Yaskawa INFORM job: OK_R2_O55B(90,0)KMOK.JBI

/JOB
//NAME OK_R2_O55B(90,0)KMOK
//POS
///NPOS 392,392,392,17,0,0
///TOOL 0
///POSTYPE PULSE
///PULSE
C00000=10240,-83405,-67778,-29541,62233,41875
C00001=74443,53482,-30,-19359,82189,66632
C00002=132592,-56559,-52251,-28632,66053,40913
C00003=129345,-24135,-32044,-25757,67809,37971
C00004=128077,-19433,-26422,-25478,66476,37777
C00005=126545,-19710,-26626,-24916,65999,37273
C00006=128077,-19433,-26422,-25478,66476,37777
C00007=128077,-19205,-24592,-25664,65564,37989
C00008=128077,-19433,-26422,-25478,66476,37777
C00009=127855,-14483,-22733,-25349,66655,37648
C00010=128077,-19433,-26422,-25478,66476,37777
C00011=128831,-22488,-30680,-25570,67657,37802
C00012=131328,-25866,-35393,-26270,69484,38362
C00013=105362,-34489,-43309,25691,63108,24690
C00014=105506,-28668,-33620,26305,60379,24076
C00015=105705,-24608,-28573,26473,59398,23909
C00016=105689,-24392,-27343,26648,58825,23753
C00017=105705,-24608,-28573,26473,59398,23909
C00018=105942,-21948,-26691,26312,59510,24040
C00019=105705,-24608,-28573,26473,59398,23909
C00020=105810,-30681,-34237,26332,59694,24030
C00021=105674,-36363,-40882,26105,60791,24250
C00022=103128,-59362,-53746,28284,58232,22422
C00023=131703,-20648,-10182,-29245,58174,41475
C00024=129196,-16533,-4757,-28754,56230,40918
C00025=126149,-3315,1827,-22038,65549,35319
C00026=126149,-2778,3575,-22172,64804,35468
C00027=126149,-3315,1827,-22038,65549,35319
C00028=124687,-3514,1666,-21646,65158,34817
C00029=126149,-3315,1827,-22038,65549,35319
C00030=126037,287,4808,-22006,65537,35277
C00031=127852,-16066,-3331,-28477,55208,40605
C00032=128831,-17793,-5581,-28669,55981,40825
C00033=131353,-23689,-16621,-28452,60169,40750
C00034=105306,-30907,-23656,28514,53942,22215
C00035=105451,-24787,-16501,28889,52781,21931
C00036=105748,-19475,-10296,29156,51720,21741
C00037=105748,-19067,-9029,29374,51220,21580
C00038=105748,-19475,-10296,29156,51720,21741
C00039=105922,-17726,-9011,29036,51756,21835
C00040=105748,-19475,-10296,29156,51720,21741
C00041=105734,-26360,-16311,29101,51869,21782
C00042=105596,-32543,-23465,28716,52996,22066
C00043=103146,-52240,-31759,31823,49615,19688
C00044=131717,-20532,-10041,-29258,58155,41487
C00045=129210,-16415,-4611,-28768,56209,40930
C00046=125726,-5717,1203,-22571,62030,35720
C00047=124600,-5859,1089,-22225,61721,35324
C00048=125726,-5717,1203,-22571,62030,35720
C00049=125726,-5303,2500,-22688,61489,35835
C00050=125726,-5717,1203,-22571,62030,35720
C00051=125653,-3254,3200,-22541,62045,35686
C00052=125726,-5717,1203,-22571,62030,35720
C00053=128784,-17293,-5015,-28681,55885,40832
C00054=131298,-23300,-16397,-28418,60205,40716
C00055=105773,-31038,-23538,28349,53659,22349
C00056=105903,-24906,-16379,28733,52505,22061
C00057=106236,-19176,-10156,28906,51612,21944
C00058=106236,-18582,-8321,29223,50886,21716
C00059=106236,-18920,-9354,29043,51293,21845
C00060=106398,-17216,-8100,28928,51328,21935
C00061=106236,-18920,-9354,29043,51293,21845
C00062=105990,-26237,-16432,28932,51901,21915
C00063=105862,-32413,-23583,28545,53028,22202
C00064=103178,-48551,-23153,33432,46714,18598
C00065=131682,-20111,-9683,-29247,58140,41477
C00066=129184,-15990,-4240,-28763,56191,40923
C00067=127040,-1088,4742,-24560,65175,37666
C00068=126467,-11690,524,-28007,54635,40139
C00069=127531,-11511,663,-28398,54998,40520
C00070=127531,-11067,1898,-28573,54527,40663
C00071=127531,-11511,663,-28398,54998,40520
C00072=127446,-9507,2221,-28343,55032,40470
C00073=127531,-11511,663,-28398,54998,40520
C00074=128904,-17444,-5156,-28721,55934,40872
C00075=131423,-23616,-17139,-28383,60508,40687
C00076=105688,-30684,-23416,28352,53783,22346
C00077=105820,-24560,-16252,28734,52622,22058
C00078=106057,-19692,-10280,29061,51509,21823
C00079=106057,-19242,-8894,29301,50963,21649
C00080=106057,-19692,-10280,29061,51509,21823
C00081=106259,-17596,-8740,28917,51554,21935
C00082=106057,-19692,-10280,29061,51509,21823
C00083=106034,-26290,-16352,28940,51819,21911
C00084=105908,-32471,-23505,28552,52945,22198
C00085=103240,-57430,-47340,29139,55590,21702
C00086=131680,-19875,-9302,-29279,58038,41504
C00087=129182,-15746,-3847,-28798,56088,40952
C00088=127763,-11793,120,-28421,55243,40554
C00089=127763,-11187,1809,-28663,54602,40747
C00090=127763,-11793,120,-28421,55243,40554
C00091=126428,-12019,-55,-27932,54786,40076
C00092=127763,-11793,120,-28421,55243,40554
C00093=127667,-9572,1845,-28358,55279,40497
C00094=127763,-11793,120,-28421,55243,40554
C00095=128878,-17535,-5369,-28685,55999,40840
C00096=131397,-24246,-19366,-28107,61425,40422
C00097=105596,-30428,-23258,28382,53845,22322
C00098=105731,-24307,-16087,28765,52679,22032
C00099=105964,-19427,-9965,29125,51490,21773
C00100=105964,-19008,-8676,29352,50979,21612
C00101=105964,-19427,-9965,29125,51490,21773
C00102=106146,-17563,-8595,28999,51530,21874
C00103=105964,-19427,-9965,29125,51490,21773
C00104=106055,-26245,-16306,28933,51808,21917
C00105=103176,-54287,-36697,30953,51210,20316
C00106=103176,-54287,-36697,30953,51210,20316
C00107=114756,-19958,-23748,4768,67559,29134
C00108=116139,-18803,-17118,-4242,63507,29437
C00109=122978,-12099,-10750,-16592,66093,31815
C00110=122978,-11495,-8359,-16737,64980,31977
C00111=122982,-12162,-10065,-16649,65658,31878
C00112=121832,-12217,-10107,-16291,65423,31469
C00113=122988,-12906,-11150,-16616,65934,31840
C00114=123134,-22680,-18382,-16732,65415,31972
C00115=117879,-24479,-16681,-8596,59721,23409
C00116=117904,-23072,-15686,-8596,59834,23409
C00117=118573,-28074,-21596,-8764,60960,23581
C00118=139843,-43230,-38559,-29857,68480,-19080
C00119=155576,-42864,-35821,-41350,65515,-28225
C00120=156680,-25452,-21834,-49402,55441,-44843
C00121=157625,-11795,-9945,-68294,73257,-47337
C00122=155300,-9623,-5312,-68606,71014,-46888
C00123=154236,-7511,-1206,-68991,69742,-46386
C00124=154236,-7054,266,-69215,69486,-46084
C00125=154236,-7511,-1206,-68991,69742,-46386
C00126=153910,-5990,11,-68964,69537,-46444
C00127=154236,-7511,-1206,-68991,69742,-46386
C00128=156732,-10707,-4701,-68974,71616,-46273
C00129=159088,-12866,-9320,-68642,73874,-46723
C00130=157785,-12020,-9831,-68356,73290,-47233
C00131=155455,-9843,-5195,-68673,71046,-46784
C00132=154312,-7370,-806,-69053,69723,-46297
C00133=154312,-6958,503,-69250,69494,-46028
C00134=154312,-7370,-806,-69053,69723,-46297
C00135=153965,-5762,476,-69025,69507,-46359
C00136=154312,-7370,-806,-69053,69723,-46297
C00137=156851,-10510,-4837,-68926,71768,-46340
C00138=159204,-12645,-9439,-68604,74024,-46790
C00139=157690,-12072,-10010,-68326,73260,-47284
C00140=155360,-9896,-5377,-68641,71015,-46835
C00141=154250,-7627,-1259,-69001,69740,-46371
C00142=154250,-7165,219,-69222,69483,-46066
C00143=154250,-7627,-1259,-69001,69740,-46371
C00144=153893,-5954,78,-68966,69513,-46438
C00145=154250,-7627,-1259,-69001,69740,-46371
C00146=156734,-10980,-5063,-68950,71650,-46310
C00147=159094,-13131,-9672,-68622,73909,-46758
C00148=157604,-12431,-10269,-68326,73193,-47285
C00149=155270,-10247,-5634,-68640,70946,-46837
C00150=154185,-8119,-1688,-68996,69699,-46385
C00151=154185,-7714,-386,-69193,69472,-46115
C00152=154185,-8119,-1688,-68996,69699,-46385
C00153=153764,-6153,-119,-68956,69433,-46463
C00154=154185,-8119,-1688,-68996,69699,-46385
C00155=156695,-11066,-5147,-68945,71627,-46318
C00156=159057,-13219,-9755,-68619,73887,-46766
C00157=157698,-12465,-10328,-68329,73262,-47279
C00158=155363,-10290,-5700,-68642,71016,-46832
C00159=154143,-7550,-1269,-68981,69685,-46406
C00160=154143,-7148,33,-69180,69456,-46136
C00161=154143,-7550,-1269,-68981,69685,-46406
C00162=153809,-5984,-19,-68952,69474,-46467
C00163=154143,-7550,-1269,-68981,69685,-46406
C00164=156735,-11186,-5208,-68955,71644,-46302
C00165=159098,-13338,-9815,-68628,73905,-46750
C00166=156103,3213,12141,-69415,68556,-43538
C00167=154648,1601,10769,-69368,67583,-43742
C00168=153106,4673,14311,-69553,66323,-43673
C00169=154059,355,8427,-69047,67491,-44191
C00170=154919,47,9463,-69374,67768,-43708
C00171=152167,817,11077,-69516,65698,-43806
C00172=152577,5510,15122,-69684,70616,-42858
C00173=152713,10209,19273,-69668,74758,-41983
C00174=154748,1711,10860,-69098,71812,-57936
C00175=156722,3942,12761,-69113,73130,-57662
C00176=156134,460,4083,-68219,69946,-45140
C00177=154681,80,6768,-68757,68248,-44508
C00178=152839,3570,11779,-69163,66517,-44175
C00179=154092,-586,6132,-68707,67871,-44613
C00180=154953,-932,7134,-69037,68144,-44129
C00181=152257,840,9559,-69164,66109,-44242
C00182=152546,4750,12892,-69392,70659,-43298
C00183=152347,7029,14931,-69460,73572,-42679
C00184=154780,436,7623,-68718,72349,-58529
C00185=156755,1502,5781,-68342,74331,-59003
C00186=156066,3482,12370,-69415,68531,-43541
C00187=154614,1870,10997,-69367,67559,-43746
C00188=153114,4686,14357,-69561,66317,-43665
C00189=154026,624,8652,-69046,67469,-44196
C00190=154884,314,9688,-69374,67743,-43712
C00191=152574,2158,12198,-69533,65964,-43752
C00192=151496,-1826,8928,-69510,65223,-43883
C00193=152752,10330,19360,-69669,74676,-41930
C00194=154713,1980,11089,-69099,71789,-57940
C00195=156684,4211,12991,-69115,73104,-57664
C00196=156120,3078,12026,-69415,68569,-43536
C00197=154664,1466,10655,-69368,67595,-43740
C00198=153101,4272,13633,-69469,66395,-43776
C00199=154076,222,8314,-69048,67503,-44190
C00200=154936,-87,9351,-69375,67779,-43705
C00201=152419,1625,11530,-69473,65914,-43837
C00202=152835,7136,16367,-69667,71654,-42618
C00203=152863,11835,20576,-69631,75787,-41730
C00204=154765,1577,10746,-69097,71825,-57934
C00205=156740,3807,12645,-69113,73143,-57660
C00206=156084,3348,12256,-69415,68544,-43539
C00207=154630,1736,10884,-69368,67571,-43744
C00208=153149,4450,14003,-69523,66373,-43704
C00209=154043,490,8540,-69046,67479,-44194
C00210=154902,181,9576,-69375,67755,-43710
C00211=152531,1941,11980,-69520,65943,-43770
C00212=152744,6177,15732,-69692,70681,-42756
C00213=152906,12246,21134,-69653,75798,-41661
C00214=154730,1846,10975,-69098,71800,-57938
C00215=156703,4077,12876,-69113,73117,-57664
C00216=148910,3102,3237,-31444,61409,-58506
C00217=134881,-38273,-33613,-7030,58257,-25285
C00218=112135,-54693,-51739,17586,56290,-4056
C00219=103817,-33181,-15280,43143,36662,33093
C00220=107418,-26920,-11084,40161,35439,34946
C00221=117558,-24459,-8743,11270,26339,51229
C00222=117529,-24457,-8742,11309,26343,51208
C00223=112868,-27530,-10869,17643,26909,47814
C00224=104598,-25779,-9605,37472,33422,36622
C00225=102251,-25540,-9311,39333,34413,35492
C00226=101145,-25457,-9112,40211,34852,34952
C00227=110637,-29640,-12060,10247,25742,51393
C00228=112099,-34921,-17271,7049,25870,53484
C00229=104953,-11353,1575,15454,55997,11022
C00230=131704,-13551,-1392,-30522,58599,57008
C00231=129362,-14151,-1850,-29808,57738,56216
C00232=125116,-13215,-2120,-23575,56441,54422
C00233=129934,-13908,-1668,-29984,57951,56409
C00234=128904,-14865,-3688,-29433,58245,55859
C00235=125052,-12029,-1213,-23540,56468,54389
C00236=124865,-5836,3553,-23405,56645,54268
C00237=124763,-3486,5457,-23358,56648,54223
C00238=128301,-14371,-2017,-29483,52718,55118
C00239=130584,-13853,-1621,-30374,53549,55940
C00240=131922,-29834,-13337,-31158,53189,56646
C00241=101101,-63378,-47161,41397,41153,33977
C00242=104308,-39459,-33280,36749,42545,36833
C00243=104497,-33395,-26443,37348,41583,36470
C00244=105232,-26009,-19438,37218,40852,36556
C00245=104776,-33046,-25034,37639,40910,36298
C00246=104569,-31396,-25208,37120,41768,36607
C00247=106202,-25772,-19324,36523,40476,36978
C00248=107261,-25140,-18860,35757,40060,37438
C00249=108104,-24816,-18601,35154,39715,37802
C00250=108611,-24652,-18486,34780,39518,38026
C00251=110769,-33421,-26459,29251,37310,41253
C00252=110982,-39482,-33293,28397,38198,41740
C00253=114569,-21613,-36743,4189,71094,21742
C00254=113623,-21477,-33729,4606,69364,21345
C00255=113177,-17466,-28904,4807,68487,21151
C00256=113244,-21406,-33755,4752,69439,21214
C00257=113428,-23529,-34032,4707,68511,21243
C00258=112388,-17537,-28888,5121,68489,20869
C00259=111067,-17855,-29089,5642,68534,20400
C00260=109895,-17947,-29146,6101,68606,19981
C00261=108779,-18084,-29248,6535,68684,19586
C00262=106055,-19215,-32051,13108,71973,13467
C00263=106183,-20073,-32808,13061,71978,13513
C00264=132180,-20263,-31618,-27417,72123,53539
C00265=129840,-20753,-29219,-26913,69821,53179
C00266=127409,-19341,-26482,-25393,67697,52783
C00267=129928,-20511,-27941,-27048,69257,53351
C00268=128899,-20993,-29537,-26589,69585,52863
C00269=127343,-18244,-25658,-25359,67726,52750
C00270=126915,-11965,-20957,-25152,67899,52540
C00271=126842,-9897,-19423,-25107,67981,52491
C00272=128299,-20899,-27421,-26008,63661,52103
C00273=130583,-20621,-29878,-26582,65870,52496
C00274=131653,-34125,-39493,-27116,65328,53027
C00275=102476,-48499,-24956,45771,36042,31536
C00276=104426,-33061,-15201,42744,36377,33351
C00277=104613,-28141,-11918,42162,36667,33686
C00278=105265,-21628,-6337,41808,36294,33919
C00279=104891,-28193,-11952,41987,36531,33799
C00280=104683,-26808,-12307,41302,37334,34174
C00281=106528,-20976,-5960,40867,35776,34509
C00282=107628,-20458,-5576,40071,35294,35008
C00283=108820,-19667,-4973,39177,34780,35558
C00284=110857,-28151,-11921,33897,31916,38728
C00285=111070,-33065,-15201,34165,31409,38600
C00286=114617,-14465,-2094,4883,53493,21055
C00287=113674,-14293,-1968,5309,53564,20668
C00288=113091,-9939,2237,5598,53256,20404
C00289=113298,-14832,-3674,5427,54358,20553
C00290=113482,-16275,-3457,5403,53475,20583
C00291=112132,-10212,2014,6030,53323,20011
C00292=110378,-10373,1991,6826,53395,19285
C00293=109598,-10558,1824,7173,53470,18965
C00294=108734,-10413,1969,7559,53529,18610
C00295=105684,-11921,-123,15049,56588,11412
C00296=106828,-11823,1079,14725,55711,11759
C00297=132184,-13138,-1076,-30660,58789,57166
C00298=129850,-13767,-1558,-29956,57927,56380
C00299=122951,-13742,-3826,-19321,56388,53347
C00300=129938,-13637,-1462,-29982,57964,56408
C00301=128912,-14594,-3483,-29430,58258,55858
C00302=126447,-11298,164,-26378,56665,55075
C00303=126149,-5151,4907,-26208,56791,54912
C00304=125929,-2212,7368,-26108,56716,54828
C00305=128294,-14104,-1815,-29475,52728,55112
C00306=130573,-13586,-1418,-30365,53557,55932
C00307=133238,-23919,-9264,-31037,58758,57600
C00308=102473,-48079,-24715,45707,36092,31571
C00309=104327,-33549,-15520,42858,36384,33282
C00310=104519,-28632,-12253,42266,36677,33624
C00311=105224,-22257,-7196,41654,36466,34003
C00312=104797,-28685,-12286,42090,36539,33738
C00313=104591,-27301,-12648,41400,37344,34114
C00314=106245,-21763,-6878,40918,36031,34468
C00315=107440,-21033,-6285,40079,35484,34993
C00316=108042,-20608,-5911,39663,35201,35253
C00317=108527,-20484,-5836,39294,34994,35480
C00318=110785,-28654,-12263,34005,31905,38669
C00319=110997,-33568,-15529,34282,31391,38533
C00320=114571,-16748,-8057,4758,55983,21151
C00321=113626,-15261,-3925,5286,54271,20683
C00322=113157,-10279,1923,5567,53271,20436
C00323=113246,-15231,-3983,5451,54348,20531
C00324=113430,-16671,-3761,5429,53463,20560
C00325=112172,-10435,1808,6013,53329,20030
C00326=110971,-10650,1676,6557,53391,19534
C00327=109888,-10687,1711,7044,53444,19090
C00328=108783,-10722,1720,7537,53520,18634
C00329=107490,-14031,-2993,12135,56057,14273
C00330=105969,-16749,-6969,14663,58214,11756
C00331=132183,-13544,-1387,-30665,58771,57170
C00332=129843,-14173,-1867,-29959,57907,56382
C00333=127984,-11675,892,-29495,56892,55850
C00334=129931,-14044,-1771,-29985,57945,56410
C00335=128902,-15001,-3790,-29434,58238,55861
C00336=127987,-10658,1630,-29475,56954,55835
C00337=127617,-5983,5353,-29317,56919,55674
C00338=127369,-2072,8539,-29220,56880,55576
C00339=128269,-14512,-2124,-29471,52703,55108
C00340=130554,-13996,-1731,-30364,53533,55929
C00341=131577,-26206,-10861,-30900,53357,56424
C00342=102457,-48470,-24939,45777,36054,31531
C00343=104393,-33223,-15307,42781,36379,33328
C00344=104581,-28304,-12029,42196,36670,33666
C00345=105392,-21894,-6807,41597,36346,34044
C00346=104859,-28357,-12063,42021,36533,33780
C00347=104652,-26971,-12421,41335,37337,34154
C00348=106233,-21462,-6455,41024,35953,34407
C00349=107408,-20797,-5933,40191,35426,34935
C00350=108113,-20379,-5618,39667,35122,35260
C00351=108958,-19959,-5342,39008,34776,35661
C00352=110833,-28319,-12035,33932,31913,38709
C00353=111045,-33232,-15311,34203,31402,38579
C00354=114601,-14596,-2193,4891,53488,21048
C00355=113657,-14424,-2067,5317,53559,20660
C00356=113150,-9858,2317,5573,53243,20434
C00357=113282,-14964,-3773,5436,54353,20545
C00358=113464,-16404,-3554,5412,53468,20575
C00359=112512,-9852,2391,5864,53243,20170
C00360=111452,-10209,2111,6342,53313,19731
C00361=110613,-10308,2046,6725,53369,19385
C00362=109868,-10452,1953,7058,53416,19076
C00363=108800,-10617,1759,7531,53547,18642
C00364=106830,-13402,-1298,13022,55655,13426
C00365=108657,-18091,-5612,12246,55609,14175
C00366=132184,-13273,-1180,-30661,58783,57167
C00367=129848,-13902,-1662,-29958,57920,56380
C00368=128083,-11609,1049,-29546,56872,55900
C00369=129936,-13773,-1565,-29983,57958,56408
C00370=128908,-14730,-3585,-29431,58252,55859
C00371=127980,-10337,2053,-29500,56867,55855
C00372=127625,-4418,6705,-29327,56900,55685
C00373=127478,-1644,8913,-29259,56911,55617
C00374=128309,-14235,-1913,-29484,52727,55120
C00375=130590,-13717,-1516,-30373,53557,55940
C00376=134769,-42597,-24032,-29392,59134,56648
C00377=134769,-42597,-24032,-29392,59134,56648
C00378=123620,-20455,-6940,-20735,55697,52350
C00379=124011,-20545,-8299,-20696,56538,52345
C00380=125642,-19637,-6354,-21475,56272,53095
C00381=123758,-19306,-6107,-20771,55803,52388
C00382=123404,-9726,1056,-20514,56199,52157
C00383=126853,-28272,-15090,-21696,57464,53362
C00384=96048,-21437,-11049,43661,69194,41767
C00385=106688,3225,9849,37167,69677,43492
C00386=109064,10097,16662,35334,71431,44136
C00387=113612,2002,4761,17318,68228,44940
C00388=111049,-2117,1500,11529,65122,43607
C00389=111472,-19995,-5761,7117,46726,41899
C00390=112310,-20229,-19914,7816,68485,44362
C00391=145371,-111898,-78356,-26837,72881,58483
BC00000=1592,516084,1075139
BC00001=71689,619329,1075149
BC00002=1593,516083,1075138
BC00003=1592,516084,1075139
BC00004=1592,516084,1075139
BC00005=1593,516084,1075138
BC00006=1592,516084,1075139
BC00007=1592,516084,1075139
BC00008=1592,516084,1075139
BC00009=1592,516084,1075139
BC00010=1592,516084,1075139
BC00011=1592,516084,1075139
BC00012=1592,516084,1075139
BC00013=1592,514680,1075139
BC00014=1592,514680,1075139
BC00015=1592,514680,1075139
BC00016=1592,514680,1075139
BC00017=1592,514680,1075139
BC00018=1592,514680,1075139
BC00019=1592,514680,1075139
BC00020=1592,514680,1075139
BC00021=1592,514680,1075139
BC00022=1592,514680,1075139
BC00023=1592,514430,1044524
BC00024=1592,514430,1044524
BC00025=1592,514430,1044524
BC00026=1592,514430,1044524
BC00027=1592,514430,1044524
BC00028=1592,514430,1044524
BC00029=1592,514430,1044524
BC00030=1592,514430,1044524
BC00031=1592,514430,1044524
BC00032=1592,514430,1044524
BC00033=1592,514430,1044524
BC00034=1592,514677,1006179
BC00035=1592,514677,1006179
BC00036=1592,514677,1006179
BC00037=1592,514677,1006179
BC00038=1592,514677,1006179
BC00039=1592,514677,1006179
BC00040=1592,514677,1006179
BC00041=1592,514677,1006179
BC00042=1592,514677,1006179
BC00043=1592,514680,1028077
BC00044=1592,514709,880841
BC00045=1592,514709,880841
BC00046=1592,514709,880841
BC00047=1592,514709,880841
BC00048=1592,514709,880841
BC00049=1592,514709,880841
BC00050=1592,514709,880841
BC00051=1592,514709,880841
BC00052=1592,514709,880841
BC00053=1592,514709,880841
BC00054=1592,514709,880841
BC00055=1592,514624,845370
BC00056=1592,514624,845370
BC00057=1592,514624,845370
BC00058=1592,514624,845370
BC00059=1592,514624,845370
BC00060=1592,514624,845370
BC00061=1592,514624,845370
BC00062=1592,514624,845370
BC00063=1592,514624,845370
BC00064=1592,514680,906645
BC00065=1592,514293,718583
BC00066=1592,514293,718583
BC00067=1592,514293,718583
BC00068=1592,514293,718583
BC00069=1592,514293,718583
BC00070=1592,514293,718583
BC00071=1592,514293,718583
BC00072=1592,514293,718583
BC00073=1592,514293,718583
BC00074=1592,514293,718583
BC00075=1592,514293,718583
BC00076=1592,514303,682531
BC00077=1592,514303,682531
BC00078=1592,514303,682531
BC00079=1592,514303,682531
BC00080=1592,514303,682531
BC00081=1592,514303,682531
BC00082=1592,514303,682531
BC00083=1592,514303,682531
BC00084=1592,514303,682531
BC00085=1592,514680,625566
BC00086=1592,514100,556875
BC00087=1592,514100,556875
BC00088=1592,514100,556875
BC00089=1592,514100,556875
BC00090=1592,514100,556875
BC00091=1592,514100,556875
BC00092=1592,514100,556875
BC00093=1592,514100,556875
BC00094=1592,514100,556875
BC00095=1592,514100,556875
BC00096=1592,514100,556875
BC00097=1592,514158,521138
BC00098=1592,514158,521138
BC00099=1592,514158,521138
BC00100=1592,514158,521138
BC00101=1592,514158,521138
BC00102=1592,514158,521138
BC00103=1592,514158,521138
BC00104=1592,514158,521138
BC00105=1592,514158,521138
BC00106=1592,514158,304508
BC00107=1592,514158,304508
BC00108=1592,514158,304508
BC00109=1592,514158,304508
BC00110=1592,514158,304508
BC00111=1592,514158,304508
BC00112=1592,514158,304508
BC00113=1592,514158,304508
BC00114=1592,514158,304508
BC00115=1592,514158,304508
BC00116=1592,514158,304508
BC00117=1592,514158,304508
BC00118=1592,507014,452875
BC00119=1592,505534,438728
BC00120=1592,503776,421929
BC00121=1592,502252,407366
BC00122=1592,502252,407366
BC00123=1592,502252,407366
BC00124=1592,502252,407366
BC00125=1592,502252,407366
BC00126=1592,502252,407366
BC00127=1592,502252,407366
BC00128=1592,502252,407366
BC00129=1592,502252,407366
BC00130=1592,502319,570498
BC00131=1592,502319,570498
BC00132=1592,502319,570498
BC00133=1592,502319,570498
BC00134=1592,502319,570498
BC00135=1592,502319,570498
BC00136=1592,502319,570498
BC00137=1592,502319,570498
BC00138=1592,502319,570498
BC00139=1592,502466,731723
BC00140=1592,502466,731723
BC00141=1592,502466,731723
BC00142=1592,502466,731723
BC00143=1592,502466,731723
BC00144=1592,502466,731723
BC00145=1592,502466,731723
BC00146=1592,502466,731723
BC00147=1592,502466,731723
BC00148=1592,502688,893934
BC00149=1592,502688,893934
BC00150=1592,502688,893934
BC00151=1592,502688,893934
BC00152=1592,502688,893934
BC00153=1592,502688,893934
BC00154=1592,502688,893934
BC00155=1592,502688,893934
BC00156=1592,502688,893934
BC00157=1592,502684,1055035
BC00158=1592,502684,1055035
BC00159=1592,502684,1055035
BC00160=1592,502684,1055035
BC00161=1592,502684,1055035
BC00162=1592,502684,1055035
BC00163=1592,502684,1055035
BC00164=1592,502684,1055035
BC00165=1592,502684,1055035
BC00166=1592,514872,787667
BC00167=1592,511098,768738
BC00168=1592,509597,761212
BC00169=1592,509588,761167
BC00170=1592,509588,761167
BC00171=1592,509588,761167
BC00172=1592,509588,761167
BC00173=1592,509588,761167
BC00174=1592,507882,765234
BC00175=1592,510298,782467
BC00176=1592,514963,1075139
BC00177=1592,511188,1075139
BC00178=1592,509679,1075136
BC00179=1592,509679,1075139
BC00180=1592,509679,1075139
BC00181=1593,509679,1075133
BC00182=1593,509679,1075133
BC00183=1593,509679,1075133
BC00184=1592,507972,1075139
BC00185=1592,510389,1075139
BC00186=1592,514782,464256
BC00187=1592,511008,445327
BC00188=1592,509498,437756
BC00189=1592,509498,437756
BC00190=1592,509498,437756
BC00191=1592,509498,437756
BC00192=1592,509498,437756
BC00193=1592,509498,437756
BC00194=1592,507791,441823
BC00195=1592,510208,459056
BC00196=1592,514917,949776
BC00197=1592,511143,930847
BC00198=1592,509633,923275
BC00199=1592,509633,923275
BC00200=1592,509633,923275
BC00201=1592,509633,923275
BC00202=1592,509633,923275
BC00203=1592,509633,923275
BC00204=1592,507927,927342
BC00205=1592,510344,944576
BC00206=1592,514827,625558
BC00207=1592,511053,606629
BC00208=1592,509543,599058
BC00209=1592,509543,599058
BC00210=1592,509543,599058
BC00211=1592,509543,599058
BC00212=1592,509543,599058
BC00213=1592,509543,599058
BC00214=1592,507836,603125
BC00215=1592,510253,620358
BC00216=1592,512810,661441
BC00217=1592,516655,723224
BC00218=1592,519659,771493
BC00219=1592,523889,839466
BC00220=1592,523889,820757
BC00221=1592,523889,813274
BC00222=1592,523889,813274
BC00223=1592,523889,813274
BC00224=1592,523889,813274
BC00225=1592,523889,813274
BC00226=1592,523889,813274
BC00227=1592,523889,813274
BC00228=1592,523889,813274
BC00229=1592,522399,939537
BC00230=1592,520013,912768
BC00231=1592,517634,894905
BC00232=1592,516682,887760
BC00233=1592,516682,887760
BC00234=1592,516682,887760
BC00235=1592,516682,887760
BC00236=1592,516682,887760
BC00237=1592,516682,887760
BC00238=1592,519458,882587
BC00239=1592,522465,899812
BC00240=1592,522465,899812
BC00241=1592,523889,1075139
BC00242=1592,523889,1075139
BC00243=1592,523889,1075139
BC00244=1592,523889,1075139
BC00245=1592,523889,1075139
BC00246=1592,523889,1075139
BC00247=1592,523889,1075139
BC00248=1592,523889,1075139
BC00249=1592,523889,1075139
BC00250=1592,523889,1075139
BC00251=1592,523889,1075139
BC00252=1592,523889,1075139
BC00253=1592,520608,1075139
BC00254=1592,515565,1075139
BC00255=1592,513548,1075139
BC00256=1592,513548,1075139
BC00257=1592,513548,1075139
BC00258=1592,513548,1075139
BC00259=1592,513548,1075139
BC00260=1592,513548,1075139
BC00261=1592,513548,1075139
BC00262=1592,517137,1075139
BC00263=1592,522490,1075139
BC00264=1592,520104,1075139
BC00265=1592,517724,1075139
BC00266=1592,516772,1075139
BC00267=1592,516772,1075139
BC00268=1592,516772,1075139
BC00269=1592,516772,1075139
BC00270=1592,516772,1075139
BC00271=1592,516772,1075139
BC00272=1592,519701,1075139
BC00273=1592,522708,1075139
BC00274=1592,522708,1075139
BC00275=1592,523889,516055
BC00276=1592,523889,516055
BC00277=1592,523889,497346
BC00278=1592,523889,489863
BC00279=1592,523889,489863
BC00280=1592,523889,489863
BC00281=1592,523889,489863
BC00282=1592,523889,489863
BC00283=1592,523889,489863
BC00284=1592,523889,497359
BC00285=1592,523889,516067
BC00286=1592,520427,616172
BC00287=1592,515385,597246
BC00288=1592,513368,589676
BC00289=1592,513368,589676
BC00290=1592,513368,589676
BC00291=1592,513368,589676
BC00292=1592,513368,589676
BC00293=1592,513368,589676
BC00294=1592,513368,589676
BC00295=1592,516956,597203
BC00296=1592,522309,616126
BC00297=1592,519923,589356
BC00298=1592,517544,571494
BC00299=1592,516592,564349
BC00300=1592,516592,564349
BC00301=1592,516592,564349
BC00302=1592,516592,564349
BC00303=1592,516592,564349
BC00304=1593,516592,564346
BC00305=1592,518754,559173
BC00306=1592,521761,576398
BC00307=1592,519923,589356
BC00308=1592,523889,1001575
BC00309=1592,523889,1001575
BC00310=1592,523889,982866
BC00311=1592,523889,975382
BC00312=1592,523889,975382
BC00313=1592,523889,975382
BC00314=1592,523889,975382
BC00315=1592,523889,975382
BC00316=1592,523889,975382
BC00317=1592,523889,975382
BC00318=1592,523889,982878
BC00319=1592,523889,1001587
BC00320=1592,520563,1075139
BC00321=1592,515520,1075139
BC00322=1592,513503,1075139
BC00323=1592,513503,1075139
BC00324=1592,513503,1075139
BC00325=1592,513503,1075139
BC00326=1592,513503,1075139
BC00327=1592,513503,1075139
BC00328=1592,513503,1075139
BC00329=1592,517092,1075139
BC00330=1592,522444,1075139
BC00331=1592,520059,1074876
BC00332=1592,517679,1057014
BC00333=1592,516727,1049869
BC00334=1592,516727,1049869
BC00335=1592,516727,1049869
BC00336=1592,516727,1049869
BC00337=1592,516727,1049869
BC00338=1592,516727,1049869
BC00339=1592,518272,1044690
BC00340=1592,521278,1061916
BC00341=1592,521278,1061916
BC00342=1592,523889,677357
BC00343=1592,523889,677357
BC00344=1592,523889,658648
BC00345=1592,523889,651165
BC00346=1592,523889,651165
BC00347=1592,523889,651165
BC00348=1592,523889,651165
BC00349=1592,523889,651165
BC00350=1592,523889,651165
BC00351=1592,523889,651165
BC00352=1592,523889,658661
BC00353=1592,523889,677369
BC00354=1592,520472,777474
BC00355=1592,515430,758548
BC00356=1592,513413,750978
BC00357=1592,513413,750978
BC00358=1592,513413,750978
BC00359=1592,513413,750978
BC00360=1592,513413,750978
BC00361=1592,513413,750978
BC00362=1592,513413,750978
BC00363=1592,513413,750978
BC00364=1592,517001,758505
BC00365=1592,517001,758505
BC00366=1592,519968,750659
BC00367=1592,517589,732796
BC00368=1592,516637,725651
BC00369=1592,516637,725651
BC00370=1592,516637,725651
BC00371=1592,516637,725651
BC00372=1592,516637,725651
BC00373=1592,516637,725651
BC00374=1592,519566,720479
BC00375=1592,522573,737704
BC00376=1592,521809,741503
BC00377=1592,508932,346542
BC00378=1592,508932,346542
BC00379=1592,508932,346542
BC00380=1592,508932,346542
BC00381=1592,508932,346542
BC00382=1592,508932,346542
BC00383=1592,508932,346542
BC00384=1592,508932,346542
BC00385=1592,508932,346542
BC00386=1592,508932,346542
BC00387=1592,508932,346542
BC00388=1592,508932,346542
BC00389=1592,508932,346542
BC00390=1592,508932,346542
BC00391=1592,519968,750659
EC00000=-798156,-183832
EC00001=-798155,-183833
EC00002=-798153,-183834
EC00003=-798156,-183832
EC00004=-798156,-183832
EC00005=-798155,-183832
EC00006=-798156,-183832
EC00007=-798156,-183832
EC00008=-798156,-183832
EC00009=-798156,-183832
EC00010=-798156,-183832
EC00011=-798156,-183832
EC00012=-798156,-183832
EC00013=-798156,-183832
EC00014=-798156,-183832
EC00015=-798156,-183832
EC00016=-798156,-183832
EC00017=-798156,-183832
EC00018=-798156,-183832
EC00019=-798156,-183832
EC00020=-798156,-183832
EC00021=-798156,-183832
EC00022=-798156,-183832
EC00023=-798156,-183832
EC00024=-798156,-183832
EC00025=-798156,-183832
EC00026=-798156,-183832
EC00027=-798156,-183832
EC00028=-798156,-183832
EC00029=-798156,-183832
EC00030=-798156,-183832
EC00031=-798156,-183832
EC00032=-798156,-183832
EC00033=-798156,-183832
EC00034=-798156,-183832
EC00035=-798156,-183832
EC00036=-798156,-183832
EC00037=-798156,-183832
EC00038=-798156,-183832
EC00039=-798156,-183832
EC00040=-798156,-183832
EC00041=-798156,-183832
EC00042=-798156,-183832
EC00043=-798156,-183832
EC00044=-798156,-183832
EC00045=-798156,-183832
EC00046=-798156,-183832
EC00047=-798156,-183832
EC00048=-798156,-183832
EC00049=-798156,-183832
EC00050=-798156,-183832
EC00051=-798156,-183832
EC00052=-798156,-183832
EC00053=-798156,-183832
EC00054=-798156,-183832
EC00055=-798156,-183832
EC00056=-798156,-183832
EC00057=-798156,-183832
EC00058=-798156,-183832
EC00059=-798156,-183832
EC00060=-798156,-183832
EC00061=-798156,-183832
EC00062=-798156,-183832
EC00063=-798156,-183832
EC00064=-798156,-183832
EC00065=-798156,-183832
EC00066=-798156,-183832
EC00067=-798156,-183832
EC00068=-798156,-183832
EC00069=-798156,-183832
EC00070=-798156,-183832
EC00071=-798156,-183832
EC00072=-798156,-183832
EC00073=-798156,-183832
EC00074=-798156,-183832
EC00075=-798156,-183832
EC00076=-798156,-183832
EC00077=-798156,-183832
EC00078=-798156,-183832
EC00079=-798156,-183832
EC00080=-798156,-183832
EC00081=-798156,-183832
EC00082=-798156,-183832
EC00083=-798156,-183832
EC00084=-798156,-183832
EC00085=-798156,-183832
EC00086=-798156,-183832
EC00087=-798156,-183832
EC00088=-798156,-183832
EC00089=-798156,-183832
EC00090=-798156,-183832
EC00091=-798156,-183832
EC00092=-798156,-183832
EC00093=-798156,-183832
EC00094=-798156,-183832
EC00095=-798156,-183832
EC00096=-798156,-183832
EC00097=-798156,-183832
EC00098=-798156,-183832
EC00099=-798156,-183832
EC00100=-798156,-183832
EC00101=-798156,-183832
EC00102=-798156,-183832
EC00103=-798156,-183832
EC00104=-798156,-183832
EC00105=-798156,-183832
EC00106=-798156,-183832
EC00107=-798156,-183832
EC00108=-798156,-183832
EC00109=-798156,-183832
EC00110=-798156,-183832
EC00111=-798156,-183832
EC00112=-798156,-183832
EC00113=-798156,-183832
EC00114=-798156,-183832
EC00115=-798156,-183832
EC00116=-798156,-183832
EC00117=-798156,-183832
EC00118=-798156,-183832
EC00119=-798156,-183832
EC00120=-798156,-183832
EC00121=-798156,-183832
EC00122=-798156,-183832
EC00123=-798156,-183832
EC00124=-798156,-183832
EC00125=-798156,-183832
EC00126=-798156,-183832
EC00127=-798156,-183832
EC00128=-798156,-183832
EC00129=-798156,-183832
EC00130=-798156,-183832
EC00131=-798156,-183832
EC00132=-798156,-183832
EC00133=-798156,-183832
EC00134=-798156,-183832
EC00135=-798156,-183832
EC00136=-798156,-183832
EC00137=-798156,-183832
EC00138=-798156,-183832
EC00139=-798156,-183832
EC00140=-798156,-183832
EC00141=-798156,-183832
EC00142=-798156,-183832
EC00143=-798156,-183832
EC00144=-798156,-183832
EC00145=-798156,-183832
EC00146=-798156,-183832
EC00147=-798156,-183832
EC00148=-798156,-183832
EC00149=-798156,-183832
EC00150=-798156,-183832
EC00151=-798156,-183832
EC00152=-798156,-183832
EC00153=-798156,-183832
EC00154=-798156,-183832
EC00155=-798156,-183832
EC00156=-798156,-183832
EC00157=-798156,-183832
EC00158=-798156,-183832
EC00159=-798156,-183832
EC00160=-798156,-183832
EC00161=-798156,-183832
EC00162=-798156,-183832
EC00163=-798156,-183832
EC00164=-798156,-183832
EC00165=-798156,-183832
EC00166=-798156,-183832
EC00167=-798156,-183832
EC00168=-798156,-183832
EC00169=-798156,-183832
EC00170=-798156,-183832
EC00171=-798156,-183832
EC00172=-798156,-183832
EC00173=-798156,-183832
EC00174=-798156,-183832
EC00175=-798156,-183832
EC00176=-798156,-183832
EC00177=-798156,-183832
EC00178=-798155,-183832
EC00179=-798156,-183832
EC00180=-798156,-183832
EC00181=-798154,-183833
EC00182=-798154,-183833
EC00183=-798154,-183833
EC00184=-798156,-183832
EC00185=-798156,-183832
EC00186=-798156,-183832
EC00187=-798156,-183832
EC00188=-798156,-183832
EC00189=-798156,-183832
EC00190=-798156,-183832
EC00191=-798156,-183832
EC00192=-798156,-183832
EC00193=-798156,-183832
EC00194=-798156,-183832
EC00195=-798156,-183832
EC00196=-798156,-183832
EC00197=-798156,-183832
EC00198=-798156,-183832
EC00199=-798156,-183832
EC00200=-798156,-183832
EC00201=-798156,-183832
EC00202=-798156,-183832
EC00203=-798156,-183832
EC00204=-798156,-183832
EC00205=-798156,-183832
EC00206=-798156,-183832
EC00207=-798156,-183832
EC00208=-798156,-183832
EC00209=-798156,-183832
EC00210=-798156,-183832
EC00211=-798156,-183832
EC00212=-798156,-183832
EC00213=-798156,-183832
EC00214=-798156,-183832
EC00215=-798156,-183832
EC00216=-798156,-183832
EC00217=-798156,-183832
EC00218=-798156,-183832
EC00219=-798156,-183832
EC00220=-798156,-183832
EC00221=-798156,-183832
EC00222=-798156,-183832
EC00223=-798156,-183832
EC00224=-798156,-183832
EC00225=-798156,-183832
EC00226=-798156,-183832
EC00227=-798154,-183835
EC00228=-798156,-183832
EC00229=-798156,-183832
EC00230=-798156,-183832
EC00231=-798156,-183832
EC00232=-798156,-183832
EC00233=-798156,-183832
EC00234=-798156,-183832
EC00235=-798156,-183832
EC00236=-798156,-183832
EC00237=-798156,-183832
EC00238=-798156,-183832
EC00239=-798156,-183832
EC00240=-798156,-183832
EC00241=-798156,-183832
EC00242=-798156,-183832
EC00243=-798156,-183832
EC00244=-798156,-183832
EC00245=-798156,-183832
EC00246=-798156,-183832
EC00247=-798156,-183832
EC00248=-798156,-183832
EC00249=-798156,-183832
EC00250=-798156,-183832
EC00251=-798156,-183832
EC00252=-798156,-183832
EC00253=-798156,-183832
EC00254=-798156,-183832
EC00255=-798156,-183832
EC00256=-798156,-183832
EC00257=-798156,-183832
EC00258=-798156,-183832
EC00259=-798156,-183832
EC00260=-798156,-183832
EC00261=-798156,-183832
EC00262=-798156,-183832
EC00263=-798156,-183832
EC00264=-798156,-183832
EC00265=-798156,-183832
EC00266=-798156,-183832
EC00267=-798156,-183832
EC00268=-798156,-183832
EC00269=-798156,-183832
EC00270=-798156,-183832
EC00271=-798156,-183832
EC00272=-798156,-183832
EC00273=-798156,-183832
EC00274=-798156,-183832
EC00275=-798156,-183832
EC00276=-798156,-183832
EC00277=-798156,-183832
EC00278=-798156,-183832
EC00279=-798156,-183832
EC00280=-798156,-183832
EC00281=-798156,-183832
EC00282=-798156,-183832
EC00283=-798156,-183832
EC00284=-798156,-183832
EC00285=-798156,-183832
EC00286=-798156,-183832
EC00287=-798156,-183832
EC00288=-798156,-183832
EC00289=-798156,-183832
EC00290=-798156,-183832
EC00291=-798156,-183832
EC00292=-798156,-183832
EC00293=-798156,-183832
EC00294=-798156,-183832
EC00295=-798156,-183832
EC00296=-798156,-183832
EC00297=-798156,-183832
EC00298=-798156,-183832
EC00299=-798156,-183832
EC00300=-798156,-183832
EC00301=-798156,-183832
EC00302=-798156,-183832
EC00303=-798156,-183832
EC00304=-798155,-183832
EC00305=-798156,-183832
EC00306=-798156,-183832
EC00307=-798156,-183832
EC00308=-798156,-183832
EC00309=-798156,-183832
EC00310=-798156,-183832
EC00311=-798156,-183832
EC00312=-798156,-183832
EC00313=-798156,-183832
EC00314=-798156,-183832
EC00315=-798156,-183832
EC00316=-798156,-183832
EC00317=-798156,-183832
EC00318=-798156,-183832
EC00319=-798156,-183832
EC00320=-798156,-183832
EC00321=-798156,-183832
EC00322=-798156,-183832
EC00323=-798156,-183832
EC00324=-798156,-183832
EC00325=-798156,-183832
EC00326=-798156,-183832
EC00327=-798156,-183832
EC00328=-798156,-183832
EC00329=-798156,-183832
EC00330=-798156,-183832
EC00331=-798156,-183832
EC00332=-798156,-183832
EC00333=-798156,-183832
EC00334=-798156,-183832
EC00335=-798156,-183832
EC00336=-798156,-183832
EC00337=-798156,-183832
EC00338=-798156,-183832
EC00339=-798156,-183832
EC00340=-798156,-183832
EC00341=-798156,-183832
EC00342=-798156,-183832
EC00343=-798156,-183832
EC00344=-798156,-183832
EC00345=-798156,-183832
EC00346=-798156,-183832
EC00347=-798156,-183832
EC00348=-798156,-183832
EC00349=-798156,-183832
EC00350=-798156,-183832
EC00351=-798156,-183832
EC00352=-798156,-183832
EC00353=-798156,-183832
EC00354=-798156,-183832
EC00355=-798156,-183832
EC00356=-798156,-183832
EC00357=-798156,-183832
EC00358=-798156,-183832
EC00359=-798156,-183832
EC00360=-798156,-183832
EC00361=-798156,-183832
EC00362=-798156,-183832
EC00363=-798156,-183832
EC00364=-798156,-183832
EC00365=-798156,-183832
EC00366=-798156,-183832
EC00367=-798156,-183832
EC00368=-798156,-183832
EC00369=-798156,-183832
EC00370=-798156,-183832
EC00371=-798156,-183832
EC00372=-798156,-183832
EC00373=-798156,-183832
EC00374=-798156,-183832
EC00375=-798156,-183832
EC00376=-798156,-183832
EC00377=-798156,-183832
EC00378=-798156,-183832
EC00379=-798156,-183832
EC00380=-798156,-183832
EC00381=-798156,-183832
EC00382=-798156,-183832
EC00383=-798156,-183832
EC00384=-798156,-183832
EC00385=-798156,-183832
EC00386=-798156,-183832
EC00387=-798156,-183832
EC00388=-798156,-183832
EC00389=-798156,-183832
EC00390=-798156,-183832
EC00391=-798156,-183832
///POSTYPE BASE
///RECTAN
///RCONF 0,0,0,0,1,0,0,0,0,0,0,0,0,0,0,0,0,0,0,0,0,0,0,0
P00006=2.006,1.622,-0.565,0.0000,0.0000,0.0000
P00021=0.073,2.058,-0.109,0.0000,0.0000,0.0000
P00022=2.006,1.622,-0.565,0.0000,0.0000,0.0000
///RCONF 0,0,0,0,0,0,0,0,0,0,0,0,0,0,0,0,0,0,0,0,0,0,0,0
P00023=-2.957,-4.083,2.762,0.0000,0.0000,0.0000
P00031=-0.170,0.039,-0.647,0.0000,0.0000,0.0000
P00032=-0.423,0.157,3.222,0.0000,0.0000,0.0000
P00033=0.854,-1.099,3.047,0.0000,0.0000,0.0000
P00041=-0.109,0.014,0.966,0.0000,0.0000,0.0000
P00042=-0.220,0.371,-0.613,0.0000,0.0000,0.0000
P00043=-0.179,-5.890,-3.227,0.0000,0.0000,0.0000
P00051=-5.945,4.696,-10.293,0.0000,0.0000,0.0000
P00052=-0.153,5.586,-7.982,0.0000,0.0000,0.0000
P00053=0.015,-0.644,-4.942,0.0000,0.0000,0.0000
P00061=1211.499,975.999,-261.374,0.5148,35.2356,175.5099
P00062=1205.574,689.500,-262.704,0.5159,35.2461,175.5270
P00063=1197.217,207.358,-268.729,0.4863,35.2395,175.4586
P00100=-8.801,1.165,-9.977,0.0000,0.0000,0.0000
//INST
///DATE 2024/11/20 12:24
///ATTR SC,RW
///GROUP1 RB1,BS1
///GROUP2 ST1
NOP
'MUZYLO 310124
'POPRAWA I SPAWANIE
'OK_R2_o55b(90,0)
'
'Path S3809
SFTOF3D
MOVJ C00000 BC00000 VJ=100.00  +MOVJ EC00000 VJ=100.00
CALL JOB:CLEAN-R1_KM_NEW
MOVJ C00001 BC00001 VJ=100.00  +MOVJ EC00001 VJ=100.00
MOVJ C00002 BC00002 VJ=100.00  +MOVJ EC00002 VJ=100.00
MOVL C00003 BC00003 V=666.7  +MOVJ EC00003 VJ=100.00
SMOVL C00004 BC00004 V=133.3  +MOVJ EC00004
SREFP 3 C00005 BC00005  +REFP EC00005
CALL JOB:SEARCH-R1-S13D
SET P021 P006
SFTON3D P021
SMOVL C00006 BC00006 V=166.7  +MOVJ EC00006
SREFP 3 C00007 BC00007  +REFP EC00007
CALL JOB:SEARCH-R1-S13D
SET P021 P006
SFTON3D P021
SMOVL C00008 BC00008 V=166.7  +MOVJ EC00008
SREFP 3 C00009 BC00009  +REFP EC00009
CALL JOB:SEARCH-R1-S13D
SET P021 P006
SFTON3D P021
SMOVL C00010 BC00010 V=166.7  +MOVJ EC00010
MOVL C00011 BC00011 V=666.7  +MOVJ EC00011 VJ=100.00
MOVL C00012 BC00012 V=1000.0  +MOVJ EC00012 VJ=100.00
'Path S3810
SFTOF3D
MOVJ C00013 BC00013 VJ=100.00  +MOVJ EC00013 VJ=100.00
MOVL C00014 BC00014 V=666.7  +MOVJ EC00014 VJ=100.00
SMOVL C00015 BC00015 V=133.3  +MOVJ EC00015
SREFP 3 C00016 BC00016  +REFP EC00016
CALL JOB:SEARCH-R1-S13D
SET P022 P006
SFTON3D P022
SMOVL C00017 BC00017 V=166.7  +MOVJ EC00017
SREFP 3 C00018 BC00018  +REFP EC00018
CALL JOB:SEARCH-R1-S13D
SET P022 P006
SFTON3D P022
SMOVL C00019 BC00019 V=166.7  +MOVJ EC00019
MOVL C00020 BC00020 V=666.7  +MOVJ EC00020 VJ=100.00
MOVL C00021 BC00021 V=1000.0  +MOVJ EC00021 VJ=100.00
MOVJ C00022 BC00022 VJ=100.00  +MOVJ EC00022 VJ=100.00
'
'Path S3811
SFTOF3D
MOVJ C00023 BC00023 VJ=100.00  +MOVJ EC00023 VJ=100.00
MOVL C00024 BC00024 V=666.7  +MOVJ EC00024 VJ=100.00
SMOVL C00025 BC00025 V=133.3  +MOVJ EC00025
SREFP 3 C00026 BC00026  +REFP EC00026
CALL JOB:SEARCH-R1-S13D
SET P031 P006
SFTON3D P031
SMOVL C00027 BC00027 V=166.7  +MOVJ EC00027
SREFP 3 C00028 BC00028  +REFP EC00028
CALL JOB:SEARCH-R1-S13D
SET P031 P006
SFTON3D P031
SMOVL C00029 BC00029 V=166.7  +MOVJ EC00029
SREFP 3 C00030 BC00030  +REFP EC00030
CALL JOB:SEARCH-R1-S13D
SET P031 P006
SFTON3D P031
SMOVL C00031 BC00031 V=166.7  +MOVJ EC00031
MOVL C00032 BC00032 V=666.7  +MOVJ EC00032 VJ=100.00
MOVL C00033 BC00033 V=1000.0  +MOVJ EC00033 VJ=100.00
'Path S3812
SFTOF3D
MOVJ C00034 BC00034 VJ=100.00  +MOVJ EC00034 VJ=100.00
MOVL C00035 BC00035 V=666.7  +MOVJ EC00035 VJ=100.00
SMOVL C00036 BC00036 V=166.7  +MOVJ EC00036
SREFP 3 C00037 BC00037  +REFP EC00037
CALL JOB:SEARCH-R1-S13D
SET P032 P006
SFTON3D P032
SMOVL C00038 BC00038 V=166.7  +MOVJ EC00038
SREFP 3 C00039 BC00039  +REFP EC00039
CALL JOB:SEARCH-R1-S13D
SET P032 P006
SFTON3D P032
SMOVL C00040 BC00040 V=166.7  +MOVJ EC00040
MOVL C00041 BC00041 V=666.7  +MOVJ EC00041 VJ=100.00
MOVL C00042 BC00042 V=1000.0  +MOVJ EC00042 VJ=100.00
MOVJ C00043 BC00043 VJ=100.00  +MOVJ EC00043 VJ=100.00
'
'Path S3813
SFTOF3D
MOVJ C00044 BC00044 VJ=100.00  +MOVJ EC00044 VJ=100.00
MOVL C00045 BC00045 V=666.7  +MOVJ EC00045 VJ=100.00
SMOVL C00046 BC00046 V=133.3  +MOVJ EC00046
SREFP 3 C00047 BC00047  +REFP EC00047
CALL JOB:SEARCH-R1-S13D
SET P041 P006
SFTON3D P041
SMOVL C00048 BC00048 V=133.3  +MOVJ EC00048
SREFP 3 C00049 BC00049  +REFP EC00049
CALL JOB:SEARCH-R1-S13D
SET P041 P006
SFTON3D P041
SMOVL C00050 BC00050 V=133.3  +MOVJ EC00050
SREFP 3 C00051 BC00051  +REFP EC00051
CALL JOB:SEARCH-R1-S13D
SET P041 P006
SFTON3D P041
SMOVL C00052 BC00052 V=166.7  +MOVJ EC00052
MOVL C00053 BC00053 V=666.7  +MOVJ EC00053 VJ=100.00
MOVL C00054 BC00054 V=1000.0  +MOVJ EC00054 VJ=100.00
'Path S3814
SFTOF3D
MOVJ C00055 BC00055 VJ=100.00  +MOVJ EC00055 VJ=100.00
MOVL C00056 BC00056 V=666.7  +MOVJ EC00056 VJ=100.00
SMOVL C00057 BC00057 V=133.3  +MOVJ EC00057
SREFP 3 C00058 BC00058  +REFP EC00058
CALL JOB:SEARCH-R1-S13D
SET P042 P006
SFTON3D P042
SMOVL C00059 BC00059 V=166.7  +MOVJ EC00059
SREFP 3 C00060 BC00060  +REFP EC00060
CALL JOB:SEARCH-R1-S13D
SET P042 P006
SFTON3D P042
SMOVL C00061 BC00061 V=166.7  +MOVJ EC00061
MOVL C00062 BC00062 V=666.7  +MOVJ EC00062 VJ=100.00
MOVL C00063 BC00063 V=1000.0  +MOVJ EC00063 VJ=100.00
MOVJ C00064 BC00064 VJ=100.00  +MOVJ EC00064 VJ=100.00
'
'Path S3815
SFTOF3D
MOVJ C00065 BC00065 VJ=100.00  +MOVJ EC00065 VJ=100.00
MOVL C00066 BC00066 V=666.7  +MOVJ EC00066 VJ=100.00
SMOVL C00067 BC00067 V=133.3  +MOVJ EC00067
SREFP 3 C00068 BC00068  +REFP EC00068
CALL JOB:SEARCH-R1-S13D
SET P051 P006
SFTON3D P051
SMOVL C00069 BC00069 V=166.7  +MOVJ EC00069
SREFP 3 C00070 BC00070  +REFP EC00070
CALL JOB:SEARCH-R1-S13D
SET P051 P006
SFTON3D P051
SMOVL C00071 BC00071 V=166.7  +MOVJ EC00071
SREFP 3 C00072 BC00072  +REFP EC00072
CALL JOB:SEARCH-R1-S13D
SET P051 P006
SFTON3D P051
SMOVL C00073 BC00073 V=166.7  +MOVJ EC00073
MOVL C00074 BC00074 V=666.7  +MOVJ EC00074 VJ=100.00
MOVL C00075 BC00075 V=1000.0  +MOVJ EC00075 VJ=100.00
'Path S3816
SFTOF3D
MOVJ C00076 BC00076 VJ=100.00  +MOVJ EC00076 VJ=100.00
MOVL C00077 BC00077 V=666.7  +MOVJ EC00077 VJ=100.00
SMOVL C00078 BC00078 V=133.3  +MOVJ EC00078
SREFP 3 C00079 BC00079  +REFP EC00079
CALL JOB:SEARCH-R1-S13D
SET P052 P006
SFTON3D P052
SMOVL C00080 BC00080 V=166.7  +MOVJ EC00080
SREFP 3 C00081 BC00081  +REFP EC00081
CALL JOB:SEARCH-R1-S13D
SET P052 P006
SFTON3D P052
SMOVL C00082 BC00082 V=166.7  +MOVJ EC00082
MOVL C00083 BC00083 V=666.7  +MOVJ EC00083 VJ=100.00
MOVL C00084 BC00084 V=1000.0  +MOVJ EC00084 VJ=100.00
MOVJ C00085 BC00085 VJ=100.00  +MOVJ EC00085 VJ=100.00
'
'Path S3817
SFTOF3D
MOVJ C00086 BC00086 VJ=100.00  +MOVJ EC00086 VJ=100.00
MOVL C00087 BC00087 V=666.7  +MOVJ EC00087 VJ=100.00
SMOVL C00088 BC00088 V=166.7  +MOVJ EC00088
SREFP 3 C00089 BC00089  +REFP EC00089
CALL JOB:SEARCH-R1-S13D
SET P061 P006
SFTON3D P061
SMOVL C00090 BC00090 V=166.7  +MOVJ EC00090
SREFP 3 C00091 BC00091  +REFP EC00091
CALL JOB:SEARCH-R1-S13D
SET P061 P006
SFTON3D P061
SMOVL C00092 BC00092 V=166.7  +MOVJ EC00092
SREFP 3 C00093 BC00093  +REFP EC00093
CALL JOB:SEARCH-R1-S13D
SET P061 P006
SFTON3D P061
SMOVL C00094 BC00094 V=166.7  +MOVJ EC00094
MOVL C00095 BC00095 V=666.7  +MOVJ EC00095 VJ=100.00
MOVL C00096 BC00096 V=1000.0  +MOVJ EC00096 VJ=100.00
'Path S3818
SFTOF3D
MOVJ C00097 BC00097 VJ=100.00  +MOVJ EC00097 VJ=100.00
MOVL C00098 BC00098 V=666.7  +MOVJ EC00098 VJ=100.00
SMOVL C00099 BC00099 V=166.7  +MOVJ EC00099
SREFP 3 C00100 BC00100  +REFP EC00100
CALL JOB:SEARCH-R1-S13D
SET P062 P006
SFTON3D P062
SMOVL C00101 BC00101 V=166.7  +MOVJ EC00101
SREFP 3 C00102 BC00102  +REFP EC00102
CALL JOB:SEARCH-R1-S13D
SET P062 P006
SFTON3D P062
SMOVL C00103 BC00103 V=166.7  +MOVJ EC00103
SFTOF3D
MOVL C00104 BC00104 V=666.7  +MOVJ EC00104 VJ=100.00
MOVL C00105 BC00105 V=1000.0  +MOVJ EC00105 VJ=100.00
MOVJ C00106 BC00106 VJ=100.00  +MOVJ EC00106 VJ=100.00
MOVJ C00107 BC00107 VJ=100.00  +MOVJ EC00107 VJ=100.00
MOVJ C00108 BC00108 VJ=100.00  +MOVJ EC00108 VJ=100.00
SMOVL C00109 BC00109 V=100.0  +MOVJ EC00109
SREFP 3 C00110 BC00110  +REFP EC00110
CALL JOB:SEARCH-R1-S13D
SET P100 P006
SFTON3D P100
SMOVL C00111 BC00111 V=166.7  +MOVJ EC00111
SREFP 3 C00112 BC00112  +REFP EC00112
CALL JOB:SEARCH-R1-S13D
SET P100 P006
SFTON3D P100
SMOVL C00113 BC00113 V=166.7  +MOVJ EC00113
SMOVL C00114 BC00114 V=250.0  +MOVJ EC00114
SMOVL C00115 BC00115 V=133.3  +MOVJ EC00115
SREFP 3 C00116 BC00116  +REFP EC00116
CALL JOB:SEARCH-R1-S13D
SET P100 P006
SFTON3D P100
SMOVL C00117 BC00117 V=166.7  +MOVJ EC00117
SFTOF3D
MOVJ C00118 BC00118 VJ=100.00  +MOVJ EC00118 VJ=100.00
'
MOVJ C00119 BC00119 VJ=100.00  +MOVJ EC00119 VJ=100.00
MOVJ C00120 BC00120 VJ=100.00  +MOVJ EC00120 VJ=100.00
'Path S3819
SFTOF3D
MOVJ C00121 BC00121 VJ=100.00  +MOVJ EC00121 VJ=100.00
MOVL C00122 BC00122 V=400.0  +MOVJ EC00122 VJ=100.00
SMOVL C00123 BC00123 V=133.3  +MOVJ EC00123
SREFP 3 C00124 BC00124  +REFP EC00124
CALL JOB:SEARCH-R1-S13D
SET P063 P006
SFTON3D P063
SMOVL C00125 BC00125 V=166.7  +MOVJ EC00125
SREFP 3 C00126 BC00126  +REFP EC00126
CALL JOB:SEARCH-R1-S13D
SET P063 P006
SFTON3D P063
SMOVL C00127 BC00127 V=166.7  +MOVJ EC00127
MOVL C00128 BC00128 V=666.7  +MOVJ EC00128 VJ=100.00
MOVL C00129 BC00129 V=1000.0  +MOVJ EC00129 VJ=100.00
'Path S3820
SFTOF3D
MOVJ C00130 BC00130 VJ=100.00  +MOVJ EC00130 VJ=100.00
MOVL C00131 BC00131 V=666.7  +MOVJ EC00131 VJ=100.00
SMOVL C00132 BC00132 V=133.3  +MOVJ EC00132
SREFP 3 C00133 BC00133  +REFP EC00133
CALL JOB:SEARCH-R1-S13D
SET P053 P006
SFTON3D P053
SMOVL C00134 BC00134 V=133.3  +MOVJ EC00134
SREFP 3 C00135 BC00135  +REFP EC00135
CALL JOB:SEARCH-R1-S13D
SET P053 P006
SFTON3D P053
SMOVL C00136 BC00136 V=133.3  +MOVJ EC00136
MOVL C00137 BC00137 V=666.7  +MOVJ EC00137 VJ=100.00
MOVL C00138 BC00138 V=1000.0  +MOVJ EC00138 VJ=100.00
'Path S3821
SFTOF3D
MOVJ C00139 BC00139 VJ=100.00  +MOVJ EC00139 VJ=100.00
MOVL C00140 BC00140 V=400.0  +MOVJ EC00140 VJ=100.00
SMOVL C00141 BC00141 V=133.3  +MOVJ EC00141
SREFP 3 C00142 BC00142  +REFP EC00142
CALL JOB:SEARCH-R1-S13D
SET P043 P006
SFTON3D P043
SMOVL C00143 BC00143 V=166.7  +MOVJ EC00143
SREFP 3 C00144 BC00144  +REFP EC00144
CALL JOB:SEARCH-R1-S13D
SET P043 P006
SFTON3D P043
SMOVL C00145 BC00145 V=166.7  +MOVJ EC00145
MOVL C00146 BC00146 V=666.7  +MOVJ EC00146 VJ=100.00
MOVL C00147 BC00147 V=1000.0  +MOVJ EC00147 VJ=100.00
'Path S3822
SFTOF3D
MOVJ C00148 BC00148 VJ=100.00  +MOVJ EC00148 VJ=100.00
MOVL C00149 BC00149 V=666.7  +MOVJ EC00149 VJ=100.00
SMOVL C00150 BC00150 V=133.3  +MOVJ EC00150
SREFP 3 C00151 BC00151  +REFP EC00151
CALL JOB:SEARCH-R1-S13D
SET P033 P006
SFTON3D P033
SMOVL C00152 BC00152 V=166.7  +MOVJ EC00152
SREFP 3 C00153 BC00153  +REFP EC00153
CALL JOB:SEARCH-R1-S13D
SET P033 P006
SFTON3D P033
SMOVL C00154 BC00154 V=166.7  +MOVJ EC00154
MOVL C00155 BC00155 V=66.7  +MOVJ EC00155 VJ=100.00
MOVL C00156 BC00156 V=1000.0  +MOVJ EC00156 VJ=100.00
'Path S3823
SFTOF3D
MOVJ C00157 BC00157 VJ=100.00  +MOVJ EC00157 VJ=100.00
MOVL C00158 BC00158 V=666.7  +MOVJ EC00158 VJ=100.00
SMOVL C00159 BC00159 V=133.3  +MOVJ EC00159
SREFP 3 C00160 BC00160  +REFP EC00160
CALL JOB:SEARCH-R1-S13D
SET P023 P006
SFTON3D P023
SMOVL C00161 BC00161 V=133.3  +MOVJ EC00161
SREFP 3 C00162 BC00162  +REFP EC00162
CALL JOB:SEARCH-R1-S13D
SET P023 P006
SFTON3D P023
SMOVL C00163 BC00163 V=133.3  +MOVJ EC00163
MOVL C00164 BC00164 V=400.0  +MOVJ EC00164 VJ=100.00
MOVL C00165 BC00165 V=1000.0  +MOVJ EC00165 VJ=100.00
'
'
'
'Path W3824
SFTOF3D
SFTON3D P043
MOVJ C00166 BC00166 VJ=100.00  +MOVJ EC00166 VJ=100.00
SMOVL C00167 BC00167 V=400.0  +MOVJ EC00167
SMOVL C00168 BC00168 V=166.7 PL=0  +MOVJ EC00168
SREFP 1 C00169 BC00169  +REFP EC00169
SREFP 2 C00170 BC00170  +REFP EC00170
MACRO1 MJ#(0) ARGF9
ARCON
SMOVL C00171 BC00171 V=9.2  +MOVJ EC00171
SMOVL C00172 BC00172 V=9.2  +MOVJ EC00172
SMOVL C00173 BC00173 V=9.2  +MOVJ EC00173
ARCOF
SMOVL C00174 BC00174 V=400.0  +MOVJ EC00174
SMOVL C00175 BC00175 V=1000.0  +MOVJ EC00175
SFTOF3D
'Path W3825
SFTOF3D
SFTON3D P023
MOVJ C00176 BC00176 VJ=100.00  +MOVJ EC00176 VJ=100.00
SMOVL C00177 BC00177 V=400.0  +MOVJ EC00177
SMOVL C00178 BC00178 V=166.7 PL=0  +MOVJ EC00178
SREFP 1 C00179 BC00179  +REFP EC00179
SREFP 2 C00180 BC00180  +REFP EC00180
ARCON
SMOVL C00181 BC00181 V=9.2  +MOVJ EC00181
SMOVL C00182 BC00182 V=9.2  +MOVJ EC00182
SMOVL C00183 BC00183 V=9.2  +MOVJ EC00183
ARCOF
SMOVL C00184 BC00184 V=400.0  +MOVJ EC00184
SMOVL C00185 BC00185 V=1000.0  +MOVJ EC00185
SFTOF3D
'Path W3826
SFTOF3D
SFTON3D P063
MOVJ C00186 BC00186 VJ=100.00  +MOVJ EC00186 VJ=100.00
SMOVL C00187 BC00187 V=400.0  +MOVJ EC00187
SMOVL C00188 BC00188 V=166.7 PL=0  +MOVJ EC00188
SREFP 1 C00189 BC00189  +REFP EC00189
SREFP 2 C00190 BC00190  +REFP EC00190
ARCON
SMOVL C00191 BC00191 V=9.2  +MOVJ EC00191
SMOVL C00192 BC00192 V=9.2  +MOVJ EC00192
SMOVL C00193 BC00193 V=9.2  +MOVJ EC00193
ARCOF
SMOVL C00194 BC00194 V=400.0  +MOVJ EC00194
SMOVL C00195 BC00195 V=1000.0  +MOVJ EC00195
SFTOF3D
'Path W3827
SFTOF3D
SFTON3D P033
MOVJ C00196 BC00196 VJ=100.00  +MOVJ EC00196 VJ=100.00
SMOVL C00197 BC00197 V=400.0  +MOVJ EC00197
SMOVL C00198 BC00198 V=166.7 PL=0  +MOVJ EC00198
SREFP 1 C00199 BC00199  +REFP EC00199
SREFP 2 C00200 BC00200  +REFP EC00200
ARCON
SMOVL C00201 BC00201 V=9.2  +MOVJ EC00201
SMOVL C00202 BC00202 V=9.2  +MOVJ EC00202
SMOVL C00203 BC00203 V=9.2  +MOVJ EC00203
ARCOF
SMOVL C00204 BC00204 V=400.0  +MOVJ EC00204
SMOVL C00205 BC00205 V=1000.0  +MOVJ EC00205
SFTOF3D
'Path W3828
SFTOF3D
SFTON3D P053
MOVJ C00206 BC00206 VJ=100.00  +MOVJ EC00206 VJ=100.00
SMOVL C00207 BC00207 V=400.0  +MOVJ EC00207
SMOVL C00208 BC00208 V=166.7 PL=0  +MOVJ EC00208
SREFP 1 C00209 BC00209  +REFP EC00209
SREFP 2 C00210 BC00210  +REFP EC00210
ARCON
SMOVL C00211 BC00211 V=9.2  +MOVJ EC00211
SMOVL C00212 BC00212 V=9.2  +MOVJ EC00212
SMOVL C00213 BC00213 V=9.2  +MOVJ EC00213
ARCOF
SMOVL C00214 BC00214 V=400.0  +MOVJ EC00214
SMOVL C00215 BC00215 V=1000.0  +MOVJ EC00215
SFTOF3D
MOVJ C00216 BC00216 VJ=100.00  +MOVJ EC00216 VJ=100.00
MOVJ C00217 BC00217 VJ=100.00  +MOVJ EC00217 VJ=100.00
MOVJ C00218 BC00218 VJ=100.00  +MOVJ EC00218 VJ=100.00
'
'Path W3829
SFTOF3D
SFTON3D P042
MOVJ C00219 BC00219 VJ=100.00  +MOVJ EC00219 VJ=100.00
SMOVL C00220 BC00220 V=400.0  +MOVJ EC00220
SFTOF3D
SFTON3D P041
SMOVL C00221 BC00221 V=166.7  +MOVJ EC00221
ARCON
SMOVC C00222 BC00222 V=9.2  +MOVJ EC00222
SMOVC C00223 BC00223 V=9.2  +MOVJ EC00223
SMOVC C00224 BC00224 V=9.2  +MOVJ EC00224
SMOVC C00225 BC00225 V=9.2  +MOVJ EC00225
SFTON3D P042
SMOVC C00226 BC00226 V=9.2  +MOVJ EC00226
SMOVL C00227 BC00227 V=9.2  +MOVJ EC00227
ARCOF
SMOVL C00228 BC00228 V=400.0  +MOVJ EC00228
SMOVL C00229 BC00229 V=1000.0  +MOVJ EC00229
SFTOF3D
'Path W3831
SFTOF3D
SFTON3D P041
MOVJ C00230 BC00230 VJ=100.00  +MOVJ EC00230 VJ=100.00
SMOVL C00231 BC00231 V=666.7  +MOVJ EC00231
SMOVL C00232 BC00232 V=166.7 PL=0  +MOVJ EC00232
SREFP 1 C00233 BC00233  +REFP EC00233
SREFP 2 C00234 BC00234  +REFP EC00234
ARCON
SMOVL C00235 BC00235 V=9.2  +MOVJ EC00235
SMOVL C00236 BC00236 V=9.2  +MOVJ EC00236
SMOVL C00237 BC00237 V=9.2  +MOVJ EC00237
ARCOF
SMOVL C00238 BC00238 V=400.0  +MOVJ EC00238
SMOVL C00239 BC00239 V=1000.0  +MOVJ EC00239
SFTOF3D
MOVJ C00240 BC00240 VJ=100.00  +MOVJ EC00240 VJ=100.00
'
'
MOVJ C00241 BC00241 VJ=100.00  +MOVJ EC00241 VJ=100.00
'Path W3832
SFTOF3D
SFTON3D P022
MOVJ C00242 BC00242 VJ=100.00  +MOVJ EC00242 VJ=100.00
SMOVL C00243 BC00243 V=666.7  +MOVJ EC00243
SMOVL C00244 BC00244 V=166.7 PL=0  +MOVJ EC00244
SREFP 1 C00245 BC00245  +REFP EC00245
SREFP 2 C00246 BC00246  +REFP EC00246
ARCON
SMOVL C00247 BC00247 V=9.2  +MOVJ EC00247
SMOVL C00248 BC00248 V=9.2  +MOVJ EC00248
SMOVL C00249 BC00249 V=9.2  +MOVJ EC00249
SMOVL C00250 BC00250 V=9.2  +MOVJ EC00250
ARCOF
SMOVL C00251 BC00251 V=400.0  +MOVJ EC00251
SMOVL C00252 BC00252 V=1000.0  +MOVJ EC00252
SFTOF3D
'Path W3833
SFTOF3D
SFTON3D P021
MOVJ C00253 BC00253 VJ=100.00  +MOVJ EC00253 VJ=100.00
SMOVL C00254 BC00254 V=666.7  +MOVJ EC00254
SMOVL C00255 BC00255 V=166.7 PL=0  +MOVJ EC00255
SREFP 1 C00256 BC00256  +REFP EC00256
SREFP 2 C00257 BC00257  +REFP EC00257
ARCON
SMOVL C00258 BC00258 V=9.2  +MOVJ EC00258
SMOVL C00259 BC00259 V=9.2  +MOVJ EC00259
SMOVL C00260 BC00260 V=9.2  +MOVJ EC00260
SMOVL C00261 BC00261 V=9.2  +MOVJ EC00261
ARCOF
SMOVL C00262 BC00262 V=400.0  +MOVJ EC00262
SMOVL C00263 BC00263 V=1000.0  +MOVJ EC00263
SFTOF3D
'Path W3834
SFTOF3D
SFTON3D P021
MOVJ C00264 BC00264 VJ=100.00  +MOVJ EC00264 VJ=100.00
SMOVL C00265 BC00265 V=666.7  +MOVJ EC00265
SMOVL C00266 BC00266 V=166.7 PL=0  +MOVJ EC00266
SREFP 1 C00267 BC00267  +REFP EC00267
SREFP 2 C00268 BC00268  +REFP EC00268
ARCON
SMOVL C00269 BC00269 V=9.2  +MOVJ EC00269
SMOVL C00270 BC00270 V=9.2  +MOVJ EC00270
SMOVL C00271 BC00271 V=9.2  +MOVJ EC00271
ARCOF
SMOVL C00272 BC00272 V=400.0  +MOVJ EC00272
SMOVL C00273 BC00273 V=1000.0  +MOVJ EC00273
SFTOF3D
MOVJ C00274 BC00274 VJ=100.00  +MOVJ EC00274 VJ=100.00
'
'
MOVJ C00275 BC00275 VJ=100.00  +MOVJ EC00275 VJ=100.00
'Path W3835
SFTOF3D
SFTON3D P062
MOVJ C00276 BC00276 VJ=100.00  +MOVJ EC00276 VJ=100.00
SMOVL C00277 BC00277 V=666.7  +MOVJ EC00277
SMOVL C00278 BC00278 V=166.7 PL=0  +MOVJ EC00278
SREFP 1 C00279 BC00279  +REFP EC00279
SREFP 2 C00280 BC00280  +REFP EC00280
ARCON
SMOVL C00281 BC00281 V=9.2  +MOVJ EC00281
SMOVL C00282 BC00282 V=9.2  +MOVJ EC00282
SMOVL C00283 BC00283 V=9.2  +MOVJ EC00283
ARCOF
SMOVL C00284 BC00284 V=400.0  +MOVJ EC00284
SMOVL C00285 BC00285 V=1000.0  +MOVJ EC00285
SFTOF3D
'Path W3836
SFTOF3D
SFTON3D P061
MOVJ C00286 BC00286 VJ=100.00  +MOVJ EC00286 VJ=100.00
SMOVL C00287 BC00287 V=666.7  +MOVJ EC00287
SMOVL C00288 BC00288 V=166.7 PL=0  +MOVJ EC00288
SREFP 1 C00289 BC00289  +REFP EC00289
SREFP 2 C00290 BC00290  +REFP EC00290
ARCON
SMOVL C00291 BC00291 V=9.2  +MOVJ EC00291
SMOVL C00292 BC00292 V=9.2  +MOVJ EC00292
SMOVL C00293 BC00293 V=9.2  +MOVJ EC00293
SMOVL C00294 BC00294 V=9.2  +MOVJ EC00294
ARCOF
SMOVL C00295 BC00295 V=400.0  +MOVJ EC00295
SMOVL C00296 BC00296 V=1000.0  +MOVJ EC00296
SFTOF3D
'Path W3837
SFTOF3D
SFTON3D P061
MOVJ C00297 BC00297 VJ=100.00  +MOVJ EC00297 VJ=100.00
SMOVL C00298 BC00298 V=666.7  +MOVJ EC00298
SMOVL C00299 BC00299 V=166.7 PL=0  +MOVJ EC00299
SREFP 1 C00300 BC00300  +REFP EC00300
SREFP 2 C00301 BC00301  +REFP EC00301
ARCON
SMOVL C00302 BC00302 V=9.2  +MOVJ EC00302
SMOVL C00303 BC00303 V=9.2  +MOVJ EC00303
SMOVL C00304 BC00304 V=9.2  +MOVJ EC00304
ARCOF
SMOVL C00305 BC00305 V=400.0  +MOVJ EC00305
SMOVL C00306 BC00306 V=1000.0  +MOVJ EC00306
SFTOF3D
MOVJ C00307 BC00307 VJ=100.00  +MOVJ EC00307 VJ=100.00
'
'
MOVJ C00308 BC00308 VJ=100.00  +MOVJ EC00308 VJ=100.00
'Path W3838
SFTOF3D
SFTON3D P032
MOVJ C00309 BC00309 VJ=100.00  +MOVJ EC00309 VJ=100.00
SMOVL C00310 BC00310 V=666.7  +MOVJ EC00310
SMOVL C00311 BC00311 V=166.7 PL=0  +MOVJ EC00311
SREFP 1 C00312 BC00312  +REFP EC00312
SREFP 2 C00313 BC00313  +REFP EC00313
ARCON
SMOVL C00314 BC00314 V=9.2  +MOVJ EC00314
SMOVL C00315 BC00315 V=9.2  +MOVJ EC00315
SMOVL C00316 BC00316 V=9.2  +MOVJ EC00316
SMOVL C00317 BC00317 V=9.2  +MOVJ EC00317
ARCOF
SMOVL C00318 BC00318 V=400.0  +MOVJ EC00318
SMOVL C00319 BC00319 V=1000.0  +MOVJ EC00319
SFTOF3D
'Path W3839
SFTOF3D
SFTON3D P031
MOVJ C00320 BC00320 VJ=100.00  +MOVJ EC00320 VJ=100.00
SMOVL C00321 BC00321 V=666.7  +MOVJ EC00321
SMOVL C00322 BC00322 V=166.7 PL=0  +MOVJ EC00322
SREFP 1 C00323 BC00323  +REFP EC00323
SREFP 2 C00324 BC00324  +REFP EC00324
ARCON
SMOVL C00325 BC00325 V=9.2  +MOVJ EC00325
SMOVL C00326 BC00326 V=9.2  +MOVJ EC00326
SMOVL C00327 BC00327 V=9.2  +MOVJ EC00327
SMOVL C00328 BC00328 V=9.2  +MOVJ EC00328
ARCOF
SMOVL C00329 BC00329 V=400.0  +MOVJ EC00329
SMOVL C00330 BC00330 V=1000.0  +MOVJ EC00330
SFTOF3D
'Path W3840
SFTOF3D
SFTON3D P031
MOVJ C00331 BC00331 VJ=100.00  +MOVJ EC00331 VJ=100.00
SMOVL C00332 BC00332 V=666.7  +MOVJ EC00332
SMOVL C00333 BC00333 V=166.7 PL=0  +MOVJ EC00333
SREFP 1 C00334 BC00334  +REFP EC00334
SREFP 2 C00335 BC00335  +REFP EC00335
ARCON
SMOVL C00336 BC00336 V=9.2  +MOVJ EC00336
SMOVL C00337 BC00337 V=9.2  +MOVJ EC00337
SMOVL C00338 BC00338 V=9.2  +MOVJ EC00338
ARCOF
SMOVL C00339 BC00339 V=400.0  +MOVJ EC00339
SMOVL C00340 BC00340 V=1000.0  +MOVJ EC00340
SFTOF3D
MOVJ C00341 BC00341 VJ=100.00  +MOVJ EC00341 VJ=100.00
'
'
MOVJ C00342 BC00342 VJ=100.00  +MOVJ EC00342 VJ=100.00
'Path W3841
SFTOF3D
SFTON3D P052
MOVJ C00343 BC00343 VJ=100.00  +MOVJ EC00343 VJ=100.00
SMOVL C00344 BC00344 V=666.7  +MOVJ EC00344
SMOVL C00345 BC00345 V=166.7 PL=0  +MOVJ EC00345
SREFP 1 C00346 BC00346  +REFP EC00346
SREFP 2 C00347 BC00347  +REFP EC00347
ARCON
SMOVL C00348 BC00348 V=9.2  +MOVJ EC00348
SMOVL C00349 BC00349 V=9.2  +MOVJ EC00349
SMOVL C00350 BC00350 V=9.2  +MOVJ EC00350
SMOVL C00351 BC00351 V=9.2  +MOVJ EC00351
ARCOF
SMOVL C00352 BC00352 V=400.0  +MOVJ EC00352
SMOVL C00353 BC00353 V=1000.0  +MOVJ EC00353
SFTOF3D
'Path W3842
SFTOF3D
SFTON3D P051
MOVJ C00354 BC00354 VJ=100.00  +MOVJ EC00354 VJ=100.00
SMOVL C00355 BC00355 V=666.7  +MOVJ EC00355
SMOVL C00356 BC00356 V=166.7 PL=0  +MOVJ EC00356
SREFP 1 C00357 BC00357  +REFP EC00357
SREFP 2 C00358 BC00358  +REFP EC00358
ARCON
SMOVL C00359 BC00359 V=9.2  +MOVJ EC00359
SMOVL C00360 BC00360 V=9.2  +MOVJ EC00360
SMOVL C00361 BC00361 V=9.2  +MOVJ EC00361
SMOVL C00362 BC00362 V=9.2  +MOVJ EC00362
SMOVL C00363 BC00363 V=9.2  +MOVJ EC00363
ARCOF
SMOVL C00364 BC00364 V=400.0  +MOVJ EC00364
SMOVL C00365 BC00365 V=1000.0  +MOVJ EC00365
SFTOF3D
'Path W3843
SFTOF3D
SFTON3D P051
MOVJ C00366 BC00366 VJ=100.00  +MOVJ EC00366 VJ=100.00
SMOVL C00367 BC00367 V=666.7  +MOVJ EC00367
SMOVL C00368 BC00368 V=166.7 PL=0  +MOVJ EC00368
SREFP 1 C00369 BC00369  +REFP EC00369
SREFP 2 C00370 BC00370  +REFP EC00370
ARCON
SMOVL C00371 BC00371 V=9.2  +MOVJ EC00371
SMOVL C00372 BC00372 V=9.2  +MOVJ EC00372
SMOVL C00373 BC00373 V=9.2  +MOVJ EC00373
ARCOF
SMOVL C00374 BC00374 V=400.0  +MOVJ EC00374
SMOVL C00375 BC00375 V=1000.0  +MOVJ EC00375
SFTOF3D
MOVJ C00376 BC00376 VJ=100.00  +MOVJ EC00376 VJ=100.00
MOVJ C00377 BC00377 VJ=100.00  +MOVJ EC00377 VJ=100.00
SFTON3D P100
SMOVL C00378 BC00378 V=166.7 PL=0  +MOVJ EC00378
SREFP 1 C00379 BC00379  +REFP EC00379
SREFP 2 C00380 BC00380  +REFP EC00380
ARCON
SWVON WEV#(102)
SMOVL C00381 BC00381 V=7.5  +MOVJ EC00381
SMOVL C00382 BC00382 V=7.5  +MOVJ EC00382
ARCOF
SWVOF
SMOVL C00383 BC00383 V=250.0  +MOVJ EC00383
SMOVL C00384 BC00384 V=250.0  +MOVJ EC00384
SMOVL C00385 BC00385 V=333.3  +MOVJ EC00385
SFTON3D P100
MACRO1 MJ#(0) ARGF14
SMOVL C00386 BC00386 V=133.3  +MOVJ EC00386
ARCON
SWVON WEV#(66)
SMOVL C00387 BC00387 V=10.8  +MOVJ EC00387
SMOVL C00388 BC00388 V=10.8  +MOVJ EC00388
SMOVL C00389 BC00389 V=10.8  +MOVJ EC00389
ARCOF
SWVOF
SFTOF3D
SMOVL C00390 BC00390 V=333.3  +MOVJ EC00390
MOVJ C00391 BC00391 VJ=100.00  +MOVJ EC00391 VJ=100.00
'
END
